(* CODESYS project Flight Simulator.project

Project tree, tasks and I/O mapping:
  PLC : HX-CP1S08, Hitachi Industrial Equipment Systems Co., Ltd., order no. HX-CP1S08, version 3.5.8.24
      settings: IP Address = '192.168.1.1'
    application Application
      libraries: Unit Conversion Interfaces, * (Intern); Standard, * (System); VisuDialogs, * (System); CAA Device Diagnosis, 3.5.4.0 (CAA Technical Workgroup); CAA Net Base Services, 3.5.8.10 (CAA Technical Workgroup); NetVarUdp, 3.5.17.0 (System); PRO JSON, 1.0.0.13 (Pro Electric)
      task Task (cyclic, interval t#20ms, priority 1, watchdog t#100ms x 1) calls MotionTest4_6Servos, TcpClient
      task EtherCAT_Task (cyclic, interval t#8ms, priority 1) calls nothing
      task VISU_TASK (cyclic, interval 100 ms, priority 31) calls VisuElems.Visu_Prg
      Symbols
      program OPC [ST]
      global variables GVL
      program stoplicht [LD]
      program MotionTest1_1Servo [FBD]
      program MotionTest3_1Servo [ST]
      program MotionTest2_1Servo [ST]
      program MotionTest3_2Servos [ST]
      program MotionTest1_2Servos [FBD]
      program MotionTest3_6Servos [ST]
      program MotionTest4_6Servos [ST]
      visualisation Main
      global variables gvlSetting
      data type ServoData
      program TcpClient [ST]
    Basic : Basic, Hitachi-IES, version 3.5.8.20
      _16_Digital_Input : 16 Digital Input, Hitachi-IES, version 3.4.0.0
          unmapped channels: ReserveWord0Type, ReserveWord0Type, ReserveWord0Type
      _16_Digital_Output : 16 Digital Output, Hitachi-IES, version 3.4.0.0
          output Application.GVL.stopLichtGroen : BOOL  // ReserveWord0Type.Bit0
          output Application.GVL.stopLichtGeel : BOOL  // ReserveWord0Type.Bit1
          output Application.GVL.stopLichtRood : BOOL  // ReserveWord0Type.Bit2
          unmapped channels: ReserveWord0Type, ReserveWord0Type, ReserveWord0Type
      _16_Digital_Input_1 : 16 Digital Input, Hitachi-IES, version 3.4.0.0
          unmapped channels: ReserveWord0Type, ReserveWord0Type, ReserveWord0Type
      _16_Digital_Output_1 : 16 Digital Output, Hitachi-IES, version 3.4.0.0
          unmapped channels: ReserveWord0Type, ReserveWord0Type, ReserveWord0Type
      <Empty>
      <Empty>
      <Empty>
      <Empty>
      <Empty>
      <Empty>
      <Empty>
    EtherCAT_Master : EtherCAT Master, Festo, version 3.5.16.43
        settings: MasterUseLRW = False; SlaveAutoRestart = True; NetworkName = 'eth2'; NetworkName = "eth2"; SelectNetworkByName = False; EnableTaskMessage = False; SrcAddress1 = 42135; SrcAddress2 = 3137775364; EnableSecondAdapter = False; SrcAddress = [16#A4,16#97,16#BB,16#06,16#A7,16#04]; NetworkName = 'eth2'; NetworkName = "eth2"; SelectNetworkByName = False
      servo_drive_1 : CMMT-AS (point to point), Festo, order no. 5340819, 534082x, 813335x, version 3.5.16.41
          settings: EnableExpertSettings = True; Watchdog register 0400 = 2498; Watchdog register 0410 = 3000; Watchdog register 0420 = 1000; Physical Address of the Slave = 1001; FMMU.Global Start Address = 16#02000000; FMMU.Physical Start Address = 16#1000; FMMU.Access = 16#02; FMMU.Global Start Address = 16#01000000; FMMU.Physical Start Address = 16#1100; FMMU.Access = 16#01; FMMU.Global Start Address = 16#00080000; FMMU.Physical Start Address = 16#080D; FMMU.Access = 16#01; DC sync0 cycletime = 8000; DC enable = 1; DC sync0 enable = 1; DC sync0 shift time = 0; DC sync1 cycletime = 8000; DC sync1 enable = 0; DC sync1 factor = 'x 1'; DC sync1 shift time = 0
          unmapped channels: Controlword, Modes of operation, Target position, Profile velocity, Target velocity, Target torque, Velocity offset, Torque offset, ---, Statusword, Modes of operation display, Position actual value, Velocity actual value, Torque actual value, Multiturns actual value, ---
      servo_drive_2 : CMMT-AS (point to point), Festo, order no. 5340819, 534082x, 813335x, version 3.5.16.41
          settings: EnableExpertSettings = True; Watchdog register 0400 = 2498; Watchdog register 0410 = 3000; Watchdog register 0420 = 1000; Physical Address of the Slave = 1002; AutoIncr Address of the Slave = 4294967295; FMMU.Global Start Address = 16#02000018; FMMU.Physical Start Address = 16#1000; FMMU.Access = 16#02; FMMU.Global Start Address = 16#01000012; FMMU.Physical Start Address = 16#1100; FMMU.Access = 16#01; FMMU.Global Start Address = 16#00080000; FMMU.StartBit = 1; FMMU.EndBit = 1; FMMU.Physical Start Address = 16#080D; FMMU.Access = 16#01; DC sync0 cycletime = 8000; DC enable = 1; DC sync0 enable = 1; DC sync0 shift time = 0; DC sync1 cycletime = 8000; DC sync1 enable = 0; DC sync1 factor = 'x 1'; DC sync1 shift time = 0
          unmapped channels: Controlword, Modes of operation, Target position, Profile velocity, Target velocity, Target torque, Velocity offset, Torque offset, ---, Statusword, Modes of operation display, Position actual value, Velocity actual value, Torque actual value, Multiturns actual value, ---
      servo_drive_3 : CMMT-AS (point to point), Festo, order no. 5340819, 534082x, 813335x, version 3.5.16.41
          settings: EnableExpertSettings = True; Watchdog register 0400 = 2498; Watchdog register 0410 = 3000; Watchdog register 0420 = 1000; Physical Address of the Slave = 1002; AutoIncr Address of the Slave = 4294967295; FMMU.Global Start Address = 16#02000018; FMMU.Physical Start Address = 16#1000; FMMU.Access = 16#02; FMMU.Global Start Address = 16#01000012; FMMU.Physical Start Address = 16#1100; FMMU.Access = 16#01; FMMU.Global Start Address = 16#00080000; FMMU.StartBit = 1; FMMU.EndBit = 1; FMMU.Physical Start Address = 16#080D; FMMU.Access = 16#01; DC sync0 cycletime = 8000; DC enable = 1; DC sync0 enable = 1; DC sync0 shift time = 0; DC sync1 cycletime = 8000; DC sync1 enable = 0; DC sync1 factor = 'x 1'; DC sync1 shift time = 0
          unmapped channels: Controlword, Modes of operation, Target position, Profile velocity, Target velocity, Target torque, Velocity offset, Torque offset, ---, Statusword, Modes of operation display, Position actual value, Velocity actual value, Torque actual value, Multiturns actual value, ---
      servo_drive_4 : CMMT-AS (point to point), Festo, order no. 5340819, 534082x, 813335x, version 3.5.16.41
          settings: EnableExpertSettings = True; Watchdog register 0400 = 2498; Watchdog register 0410 = 3000; Watchdog register 0420 = 1000; Physical Address of the Slave = 1002; AutoIncr Address of the Slave = 4294967295; FMMU.Global Start Address = 16#02000018; FMMU.Physical Start Address = 16#1000; FMMU.Access = 16#02; FMMU.Global Start Address = 16#01000012; FMMU.Physical Start Address = 16#1100; FMMU.Access = 16#01; FMMU.Global Start Address = 16#00080000; FMMU.StartBit = 1; FMMU.EndBit = 1; FMMU.Physical Start Address = 16#080D; FMMU.Access = 16#01; DC sync0 cycletime = 8000; DC enable = 1; DC sync0 enable = 1; DC sync0 shift time = 0; DC sync1 cycletime = 8000; DC sync1 enable = 0; DC sync1 factor = 'x 1'; DC sync1 shift time = 0
          unmapped channels: Controlword, Modes of operation, Target position, Profile velocity, Target velocity, Target torque, Velocity offset, Torque offset, ---, Statusword, Modes of operation display, Position actual value, Velocity actual value, Torque actual value, Multiturns actual value, ---
      servo_drive_5 : CMMT-AS (point to point), Festo, order no. 5340819, 534082x, 813335x, version 3.5.16.41
          settings: EnableExpertSettings = True; Watchdog register 0400 = 2498; Watchdog register 0410 = 3000; Watchdog register 0420 = 1000; Physical Address of the Slave = 1002; AutoIncr Address of the Slave = 4294967295; FMMU.Global Start Address = 16#02000018; FMMU.Physical Start Address = 16#1000; FMMU.Access = 16#02; FMMU.Global Start Address = 16#01000012; FMMU.Physical Start Address = 16#1100; FMMU.Access = 16#01; FMMU.Global Start Address = 16#00080000; FMMU.StartBit = 1; FMMU.EndBit = 1; FMMU.Physical Start Address = 16#080D; FMMU.Access = 16#01; DC sync0 cycletime = 8000; DC enable = 1; DC sync0 enable = 1; DC sync0 shift time = 0; DC sync1 cycletime = 8000; DC sync1 enable = 0; DC sync1 factor = 'x 1'; DC sync1 shift time = 0
          unmapped channels: Controlword, Modes of operation, Target position, Profile velocity, Target velocity, Target torque, Velocity offset, Torque offset, ---, Statusword, Modes of operation display, Position actual value, Velocity actual value, Torque actual value, Multiturns actual value, ---
      servo_drive_6 : CMMT-AS (point to point), Festo, order no. 5340819, 534082x, 813335x, version 3.5.16.41
          settings: EnableExpertSettings = True; Watchdog register 0400 = 2498; Watchdog register 0410 = 3000; Watchdog register 0420 = 1000; Physical Address of the Slave = 1002; AutoIncr Address of the Slave = 4294967295; FMMU.Global Start Address = 16#02000018; FMMU.Physical Start Address = 16#1000; FMMU.Access = 16#02; FMMU.Global Start Address = 16#01000012; FMMU.Physical Start Address = 16#1100; FMMU.Access = 16#01; FMMU.Global Start Address = 16#00080000; FMMU.StartBit = 1; FMMU.EndBit = 1; FMMU.Physical Start Address = 16#080D; FMMU.Access = 16#01; DC sync0 cycletime = 8000; DC enable = 1; DC sync0 enable = 1; DC sync0 shift time = 0; DC sync1 cycletime = 8000; DC sync1 enable = 0; DC sync1 factor = 'x 1'; DC sync1 shift time = 0
          unmapped channels: Controlword, Modes of operation, Target position, Profile velocity, Target velocity, Target torque, Velocity offset, Torque offset, ---, Statusword, Modes of operation display, Position actual value, Velocity actual value, Torque actual value, Multiturns actual value, ---
  Device : EHV-CPU1025, Hitachi-IES, order no. EHV-CPU1025, version 3.5.4.11
    application Application
      libraries: Standard, * (System); SysTimeRtc, 3.5.17.0 (System); CAA Net Base Services, 3.5.8.10 (CAA Technical Workgroup); PRO JSON, 1.0.0.11 (Pro Electric)
  libraries: VisuSymbols, 4.1.0.0 (System)
  function block Axis [ST]: init, isReady, setPosition, inError, getPosition, cycle, doMovement, doEnable, doReset, doDisable
  function block FlightSimulator [ST]: init, cycle, inError, safetyStop, doReset, doEnable, doDisable, doSyncMovement, doBullshit, setParameters
  text list GlobalTextList
*)

// PLC/Application/ServoData
TYPE ServoData :
STRUCT
	positions: ARRAY[1..6] OF JSONVAR;
	speeds: ARRAY[1..6] OF JSONVAR;
END_STRUCT
END_TYPE

// PLC/Application/GVL
{attribute 'qualified_only'}
VAR_GLOBAL
	stopLichtRood: BOOL;
	stopLichtGeel: BOOL;
	stopLichtGroen: BOOL;
	
	Axis: ARRAY[1..6] OF AXIS_REF_FESTO;
	resetKnop: BOOL := FALSE;
	enableKnop: BOOL := FALSE;
	nextPositionInput: REAL := 0;
	activateKnop: BOOL;
	bullshitKnop: BOOL;
	FlightSimulator: FlightSimulator;
	test: WSTRING := "Je Moeder";
	
END_VAR

// PLC/Application/gvlSetting
{attribute 'qualified_only'}
VAR_GLOBAL CONSTANT
    gc_uiPort        : UINT := 51223;
    gc_stIpAddr      : NBS.IP_ADDR := (sAddr := '145.48.203.188');
     
    gc_wMaxTelegram  : INT := 250; // Length o the telegram
END_VAR

// PLC/Application/MotionTest4_6Servos
PROGRAM MotionTest4_6Servos
VAR
	init: BOOL := TRUE;
	bullshitTimer: TON;
	iCounter : int;
END_VAR

IF init THEN
	GVL.FlightSimulator.init(
		axis1 := servo_drive_1,
		axis2 := servo_drive_2,
		axis3 := servo_drive_3,
		axis4 := servo_drive_4,
		axis5 := servo_drive_5,
		axis6 := servo_drive_6,
		servoData := tcpClient.servoData
	);
	init := FALSE;
END_IF

IF GVL.resetKnop THEN
	GVL.FlightSimulator.doReset();
END_IF

IF GVL.enableKnop THEN
	GVL.FlightSimulator.doEnable();
ELSE
	GVL.FlightSimulator.doDisable();	
END_IF

GVL.FlightSimulator.setParameters(tcpClient.servoData.positions, tcpClient.servoData.speeds);



IF GVL.activateKnop THEN
	//GVL.FlightSimulator.doSyncMovement(position := GVL.nextPositionInput);
	//GVL.FlightSimulator.setParameters(tcpClient.servoData.positions, tcpClient.servoData.speeds);
END_IF

IF GVL.bullshitKnop THEN
	IF bullshitTimer.Q THEN
		GVL.FlightSimulator.doBullshit();
	END_IF
	bullshitTimer(IN:= NOT bullshitTimer.Q, PT := T#0.333S);
END_IF

FOR iCounter := 1 TO 6 BY 1 DO
	GVL.FlightSimulator.currentPositions[iCounter].Number := GVL.FlightSimulator.axis[iCounter].getPosition();
END_FOR



GVL.FlightSimulator.cycle();

END_PROGRAM

// FlightSimulator
FUNCTION_BLOCK FlightSimulator
VAR_OUTPUT
	axis: ARRAY[1..6] OF Axis;
END_VAR
VAR
	sinValue: INT;
	servoData: REFERENCE TO ServoData;
	servoPositions : ARRAY[1..6] OF REAL;
	servoVelocities : ARRAY[1..6] OF REAL;
END_VAR
VAR_INPUT
	currentPositions : ARRAY[1..6] OF JSONVAR;
END_VAR

METHOD init : BOOL
VAR_INPUT
	axis1: REFERENCE TO AXIS_REF_FESTO;
	axis2: REFERENCE TO AXIS_REF_FESTO;
	axis3: REFERENCE TO AXIS_REF_FESTO;
	axis4: REFERENCE TO AXIS_REF_FESTO;
	axis5: REFERENCE TO AXIS_REF_FESTO;
	axis6: REFERENCE TO AXIS_REF_FESTO;
	servoData: REFERENCE TO ServoData;
END_VAR
THIS^.axis[1].init(axis1);
THIS^.axis[2].init(axis2);
THIS^.axis[3].init(axis3);
THIS^.axis[4].init(axis4);
THIS^.axis[5].init(axis5);
THIS^.axis[6].init(axis6);
THIS^.servoData REF= servoData;
END_METHOD

METHOD cycle : BOOL
VAR_INPUT
END_VAR
VAR
	iCounter: UINT;
END_VAR
// If any Axis is in error stop all axis.
IF THIS^.inError() THEN
	THIS^.safetyStop();
END_IF

FOR iCounter := 1 TO 6 BY 1 DO
	IF GVL.activateKnop THEN
		Axis[iCounter].doMovement(position := THIS^.servoPositions[iCounter], velocity := THIS^.servoVelocities[iCounter]);
	END_IF;
END_FOR

// Cycle Axis classes
FOR iCounter := 1 TO 6 BY 1 DO
	THIS^.axis[iCounter].cycle();
END_FOR
END_METHOD

METHOD inError : BOOL
VAR
	iCounter: UINT;
END_VAR
FOR iCounter := 1 TO 6 BY 1 DO
	IF THIS^.axis[iCounter].inError() THEN
		inError := TRUE;
	END_IF
END_FOR
END_METHOD

METHOD safetyStop : BOOL
VAR
	iCounter: UINT;
END_VAR
FOR iCounter := 1 TO 6 BY 1 DO
	Axis[iCounter].doDisable();
END_FOR
END_METHOD

METHOD doReset : BOOL
VAR_INPUT
END_VAR
VAR
	iCounter: UINT;
END_VAR
FOR iCounter := 1 TO 6 BY 1 DO
	Axis[iCounter].doReset();
END_FOR
END_METHOD

METHOD doEnable : BOOL
VAR_INPUT
END_VAR
VAR
	iCounter: INT;
END_VAR
FOR iCounter := 1 TO 6 BY 1 DO
	Axis[iCounter].doEnable();
END_FOR
doEnable := TRUE;
END_METHOD

METHOD doDisable : BOOL
VAR_INPUT
END_VAR
VAR
	iCounter: INT;
END_VAR
FOR iCounter := 1 TO 6 BY 1 DO
	Axis[iCounter].doDisable();
END_FOR
doDisable := TRUE;
END_METHOD

METHOD doSyncMovement : BOOL
VAR_INPUT
	position: REAL;
END_VAR
VAR
	iCounter: INT;
END_VAR
// Only do movements when drive is enabled
FOR iCounter := 1 TO 6 BY 1 DO
	THIS^.axis[iCounter].doMovement(position := position, velocity := 200);
END_FOR
DoSyncMovement := TRUE;	// return
END_METHOD

METHOD doBullshit : BOOL
VAR_INPUT
END_VAR
VAR
	iCounter: INT;
	newPosition: REAL;
END_VAR
FOR iCounter := 1 TO 6 BY 1 DO
	THIS^.sinValue := THIS^.sinValue + 15;
	newPosition := 200.0 + (200.0 * SIN(THIS^.sinValue));
	THIS^.axis[iCounter].doMovement(position := newPosition, velocity := 200);
END_FOR
END_METHOD

METHOD setParameters : BOOL
VAR
	iCounter: INT;
END_VAR
VAR_INPUT
	positions : ARRAY[1..6] OF JSONVAR;
	speeds : ARRAY[1..6] OF JSONVAR;
END_VAR
FOR iCounter := 1 TO 6 BY 1 DO
	THIS^.servoPositions[iCounter] := positions[iCounter].Number;
	THIS^.servoVelocities[iCounter] := speeds[iCounter].Number;
END_FOR
END_METHOD

END_FUNCTION_BLOCK

// Axis
FUNCTION_BLOCK Axis
VAR
	MC_Power: MC_Power_Festo;
	MC_Reset: MC_Reset_Festo;
	MC_MoveAbsolute: MC_MoveAbsolute_Festo;
	MC_ReadActualPosition: MC_ReadActualPosition_Festo;
	MC_ReadStatus: MC_ReadStatus_Festo;
	
	axis: REFERENCE TO AXIS_REF_FESTO;
	done: BOOL := FALSE;
	error: BOOL := FALSE;
	enable: BOOL := FALSE;
	activate: BOOL := FALSE;
	reset: BOOL := FALSE;
	position: REAL := 0;
	velocity: REAL := 200;
	acceleration: REAL := 5000;
	deceleration: REAL := 5000;
	jerk: REAL := 15000;
END_VAR

METHOD init : BOOL
VAR_INPUT
	axis : REFERENCE TO AXIS_REF_FESTO;
END_VAR
// This function references the servo drive to the instance of the function block.
THIS^.axis REF= axis;
END_METHOD

METHOD isReady : BOOL
VAR_INPUT
END_VAR
isReady := THIS^.done;
END_METHOD

METHOD setPosition : BOOL
VAR_INPUT
	position: REAL;
END_VAR
THIS^.position := position;
END_METHOD

METHOD inError : BOOL
VAR_INPUT
END_VAR
inError := THIS^.error;
END_METHOD

METHOD getPosition : REAL
VAR_INPUT
END_VAR
getPosition := THIS^.MC_ReadActualPosition.Position;
END_METHOD

METHOD cycle : BOOL
VAR_INPUT
END_VAR
THIS^.MC_Power(
	axis := THIS^.axis,
	enable := THIS^.enable
);

THIS^.MC_Reset(
	axis := THIS^.axis,
	Execute :=THIS^.reset
);

// Reset the reset variable
IF THIS^.MC_Reset.Done AND THIS^.reset THEN
	THIS^.reset := FALSE;
END_IF

THIS^.MC_MoveAbsolute(
	axis := THIS^.axis,
	Execute := THIS^.activate,
	ContinuousUpdate := FALSE,
	position := THIS^.position,
	velocity := THIS^.velocity,
	acceleration := THIS^.acceleration,
	deceleration := THIS^.deceleration,
	jerk := THIS^.jerk
);

// Reset the activate variable
IF THIS^.MC_MoveAbsolute.Done THEN
	THIS^.activate := FALSE;
	THIS^.done := TRUE;
END_IF

THIS^.MC_ReadActualPosition(
	axis := THIS^.axis,
	Enable := TRUE
);

THIS^.error := THIS^.MC_Power.Error OR THIS^.MC_MoveAbsolute.Error;

//MC_ReadStatus(THIS^.axis);
END_METHOD

METHOD doMovement : BOOL
VAR_INPUT
	velocity: REAL;
	position: REAL;
END_VAR
// Only do movements when drive is enabled
IF THIS^.enable THEN
	THIS^.position := position;
	THIS^.velocity := velocity;
	THIS^.activate := TRUE;
	DoMovement := TRUE;	// return
ELSE
	DoMovement := FALSE;	// return
END_IF;
END_METHOD

METHOD doEnable : BOOL
// Only allow enable when not in error
IF NOT THIS^.inError() THEN
	THIS^.enable := TRUE;
	doEnable := TRUE;
ELSE
	doEnable := FALSE;
END_IF
END_METHOD

METHOD doReset
THIS^.reset := TRUE;
END_METHOD

METHOD doDisable : BOOL
VAR_INPUT
END_VAR
// Allow disable at any time
THIS^.enable := FALSE;
doDisable := TRUE;
END_METHOD

END_FUNCTION_BLOCK

// PLC/Application/TcpClient
PROGRAM TcpClient
VAR
    fbTcpClient   : NBS.TCP_Client;
    fbTcpRead     : NBS.TCP_Read;
    fbTcpWrite    : NBS.TCP_Write;
 
	received      : STRING;
	sent          : STRING;
	parseJSON     : JSON_TO_STRUCT;
	composeJSON   : STRUCT_TO_JSON;
	servoData     : ServoData;
 
    udiVal        : UDINT;
    pudiVal       : POINTER TO BYTE;
    iIndex        : INT;
    xConnect      : BOOL;
 
    xRead         : BOOL := TRUE;
    xMissingAck   : BOOL;
    udiResult     : UDINT;
    udiLastAck    : UDINT;
    udiNow        : UDINT;
    udiRead       : UDINT;
END_VAR

fbTcpClient(xEnable := xConnect, ipAddr := gvlSetting.gc_stIpAddr, uiPort := gvlSetting.gc_uiPort, udiTimeOut := 0);

IF NOT fbTcpWrite.xBusy THEN
	IF NOT composeJSON.Busy THEN
		composeJSON(
		Execute:= TRUE,
		JSONString:= ADR(sent), 
		JSONStringSize:= SIZEOF(sent),
		JSONVars:= ADR(GVL.FlightSimulator.currentPositions),
		NumberOfVars:= SIZEOF(GVL.FlightSimulator.currentPositions) / SIZEOF(JSONVAR)
		);	
	ELSIF composeJSON.Done THEN
		fbTcpWrite(xExecute := xConnect, hConnection := fbTcpClient.hConnection, udiTimeOut := 0, szSize := SIZEOF(sent), pData := ADR(sent));
	END_IF
ELSIF fbTcpWrite.xDone THEN
	fbTcpWrite(xExecute := FALSE);
	composeJSON(Execute := FALSE);	
END_IF

IF NOT fbTcpRead.xBusy THEN
	fbTcpRead(xEnable := xRead AND xConnect, hConnection := fbTcpClient.hConnection, szSize := SIZEOF(received), pData := ADR(received), szCount => udiRead);
	IF fbTcpRead.xReady THEN
		parseJSON(	
		Execute := TRUE,
		JSONString:= ADR(received), 
		JSONStringSize:= SIZEOF(received),
		JSONVars:= ADR(servoData),
		NumberOfVars:= SIZEOF(servoData) / SIZEOF(JSONVAR)
		);
		IF parseJSON.Done THEN
			parseJSON(Execute := FALSE);
		END_IF
	END_IF
END_IF
 
IF NOT fbTcpClient.xActive AND NOT fbTcpClient.xBusy AND NOT fbTcpClient.xDone THEN
    xConnect := TRUE;
ELSIF fbTcpClient.xDone THEN
    xConnect := FALSE;
END_IF

END_PROGRAM

// PLC/Application/OPC
PROGRAM OPC
VAR
	enable : BOOL := FALSE;
	count : INT := 0;
END_VAR

IF enable THEN
	count := count + 1;
END_IF

END_PROGRAM

// PLC/Application/stoplicht
PROGRAM stoplicht
VAR
	timer_1: TON;
	timer_2: TON;
	counter_1: CTU;
END_VAR

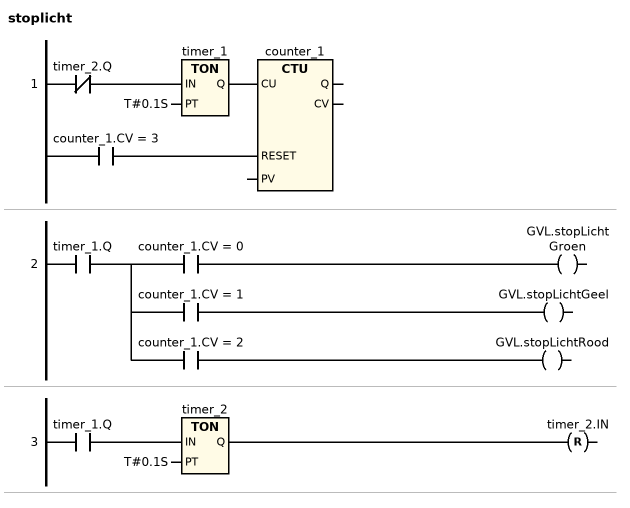
// NETWORK 1
timer_1(IN := NOT timer_2.Q, PT := T#0.1S); // TON
counter_1(CU := timer_1.Q, RESET := counter_1.CV = 3); // CTU

// NETWORK 2
GVL.stopLichtGroen := timer_1.Q AND (counter_1.CV = 0);
GVL.stopLichtGeel := timer_1.Q AND (counter_1.CV = 1);
GVL.stopLichtRood := timer_1.Q AND (counter_1.CV = 2);

// NETWORK 3
timer_2(IN := timer_1.Q, PT := T#0.1S); // TON
timer_2.IN R= timer_2.Q;

END_PROGRAM

// PLC/Application/MotionTest1_1Servo
PROGRAM MotionTest1_1Servo
VAR
	MC_Power: MC_Power_Festo;
	MC_Reset: MC_Reset_Festo;
	MC_MoveAbsolute: MC_MoveAbsolute_Festo;
	Pos: REAL := 0;
	Vel: REAL := 400;
	Acc: REAL := 5000;
	Dec: REAL := 5000;
	Jerk: REAL := 150000;
	Active: BOOL := FALSE;
	Reset: BOOL := FALSE;
	Power: BOOL := FALSE;
	Done: BOOL;
END_VAR
VAR // added by the converter: edge detectors and wires of the graphical bodies
    _w1, _w2 : BOOL;
END_VAR

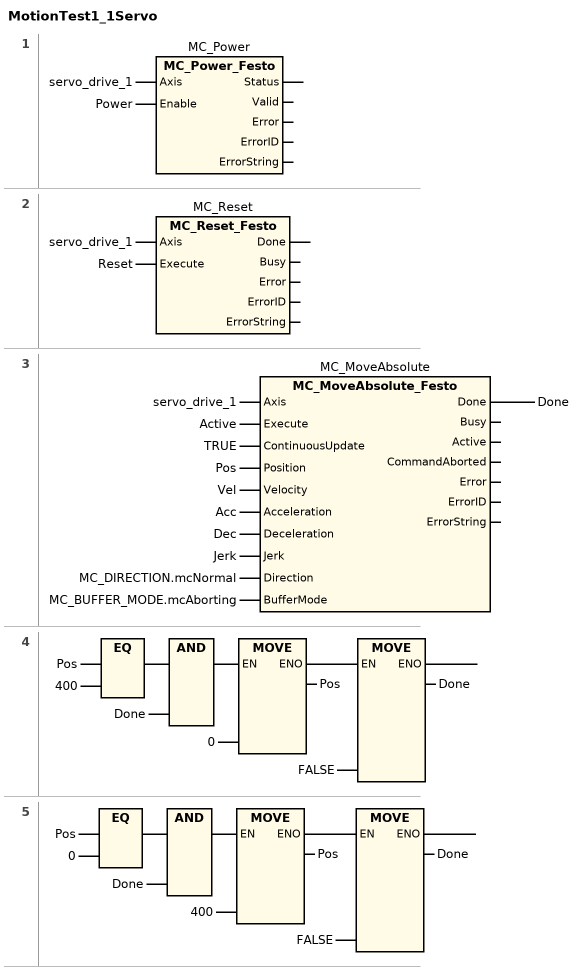
// NETWORK 1
MC_Power(Axis := servo_drive_1, Enable := Power); // MC_Power_Festo

// NETWORK 2
MC_Reset(Axis := servo_drive_1, Execute := Reset); // MC_Reset_Festo

// NETWORK 3
MC_MoveAbsolute(
    Axis := servo_drive_1,
    Execute := Active,
    ContinuousUpdate := TRUE,
    Position := Pos,
    Velocity := Vel,
    Acceleration := Acc,
    Deceleration := Dec,
    Jerk := Jerk,
    Direction := MC_DIRECTION.mcNormal,
    BufferMode := MC_BUFFER_MODE.mcAborting); // MC_MoveAbsolute_Festo
Done := MC_MoveAbsolute.Done;

// NETWORK 4
_w1 := Pos = 400 AND Done;
IF _w1 THEN Pos := 0; END_IF
IF _w1 THEN Done := FALSE; END_IF

// NETWORK 5
_w2 := Pos = 0 AND Done;
IF _w2 THEN Pos := 400; END_IF
IF _w2 THEN Done := FALSE; END_IF

END_PROGRAM

// PLC/Application/MotionTest3_1Servo
PROGRAM MotionTest3_1Servo

VAR
	Pos: REAL := 0;
	Vel: REAL := 400;
	Acc: REAL := 5000;
	Dec: REAL := 5000;
	Jerk: REAL := 150000;
	Active: BOOL := FALSE;
	Power: BOOL := FALSE;
	Done: BOOL;
	init: BOOL := TRUE;
	reset: BOOL := FALSE;
	Axis: Axis;
	inError: BOOL;
END_VAR

//MC_Power(Axis:=servo_drive_1, Enable:=Power, Error => inError);
//MC_Reset(Axis:=servo_drive_1, Execute:=reset, Error => inError);

//MC_MoveAbsolute(Axis:=servo_drive_1, Execute:=Active, ContinuousUpdate:=TRUE, Position:=Pos, Velocity:=Vel, Acceleration:=Acc, Deceleration:=Dec, Jerk:=Jerk);
IF init THEN
	Axis.init(Axis := servo_drive_1);
END_IF

IF Axis.getPosition() >= 399 THEN
	Axis.setPosition(Position := 0);
END_IF

IF Axis.getPosition() <= 1 THEN
	Axis.setPosition(Position := 400);
END_IF

Axis.cycle();

END_PROGRAM

// PLC/Application/MotionTest2_1Servo
PROGRAM MotionTest2_1Servo

VAR
	MC_Power: MC_Power_Festo;
	MC_Reset: MC_Reset_Festo;
	MC_MoveAbsolute: MC_MoveAbsolute_Festo;
	MC_ReadActualPosition: MC_ReadActualPosition_Festo;
	MC_ReadStatus: MC_ReadStatus_Festo;
	Pos: REAL := 0;
	Vel: REAL := 400;
	Acc: REAL := 5000;
	Dec: REAL := 5000;
	Jerk: REAL := 150000;
	Active: BOOL := FALSE;
	Power: BOOL := FALSE;
	Done: BOOL;
	init: BOOL := TRUE;
	reset: BOOL := FALSE;
	Axis: AXIS_REF_FESTO;
	inError: BOOL;
END_VAR

MC_Power(Axis:=servo_drive_1, Enable:=Power, Error => inError);
MC_Reset(Axis:=servo_drive_1, Execute:=reset, Error => inError);

MC_MoveAbsolute(Axis:=servo_drive_1, Execute:=Active, ContinuousUpdate:=TRUE, Position:=Pos, Velocity:=Vel, Acceleration:=Acc, Deceleration:=Dec, Jerk:=Jerk);

END_PROGRAM

// PLC/Application/MotionTest3_2Servos
PROGRAM MotionTest3_2Servos

VAR
	Pos: REAL := 0;
	Vel: REAL := 400;
	Acc: REAL := 5000;
	Dec: REAL := 5000;
	Jerk: REAL := 150000;
	Active: BOOL := FALSE;
	Power: BOOL := FALSE;
	Done: BOOL;
	init: BOOL := TRUE;
	reset: BOOL := FALSE;
	Axis2: Axis;
	Axis1: Axis;
	inError: BOOL;
END_VAR

IF init THEN
	Axis1.init(Axis := servo_drive_1);
	Axis2.init(Axis := servo_drive_2);
END_IF

IF Axis1.getPosition() >= 399 THEN
	Axis1.setPosition(Position := 0);
END_IF

IF Axis1.getPosition() <= 1 THEN
	Axis1.setPosition(Position := 400);
END_IF

IF Axis2.getPosition() >= 399 THEN
	Axis2.setPosition(Position := 0);
END_IF

IF Axis2.getPosition() <= 1 THEN
	Axis2.setPosition(Position := 400);
END_IF

Axis1.cycle();
Axis2.cycle();

END_PROGRAM

// PLC/Application/MotionTest1_2Servos
PROGRAM MotionTest1_2Servos
VAR
	MC_Power_Festo_0: MC_Power_Festo;
	MC_Reset_Festo_0: MC_Reset_Festo;
	MC_MoveAbsolute_Festo_0: MC_MoveAbsolute_Festo;
	Pos: REAL := 0;
	Vel: REAL := 400;
	Acc: REAL := 5000;
	Dec: REAL := 5000;
	Jerk: REAL := 150000;
	Active2: BOOL := FALSE;
	Active: BOOL := FALSE;
	Reset: BOOL := FALSE;
	Power: BOOL := FALSE;
	Power2: BOOL := FALSE;
	Done: BOOL;
	MC_Power_Festo_1: MC_Power_Festo;
	MC_Reset_Festo_1: MC_Reset_Festo;
	MC_MoveAbsolute_Festo_1: MC_MoveAbsolute_Festo;
END_VAR
VAR // added by the converter: edge detectors and wires of the graphical bodies
    _w1, _w2 : BOOL;
END_VAR

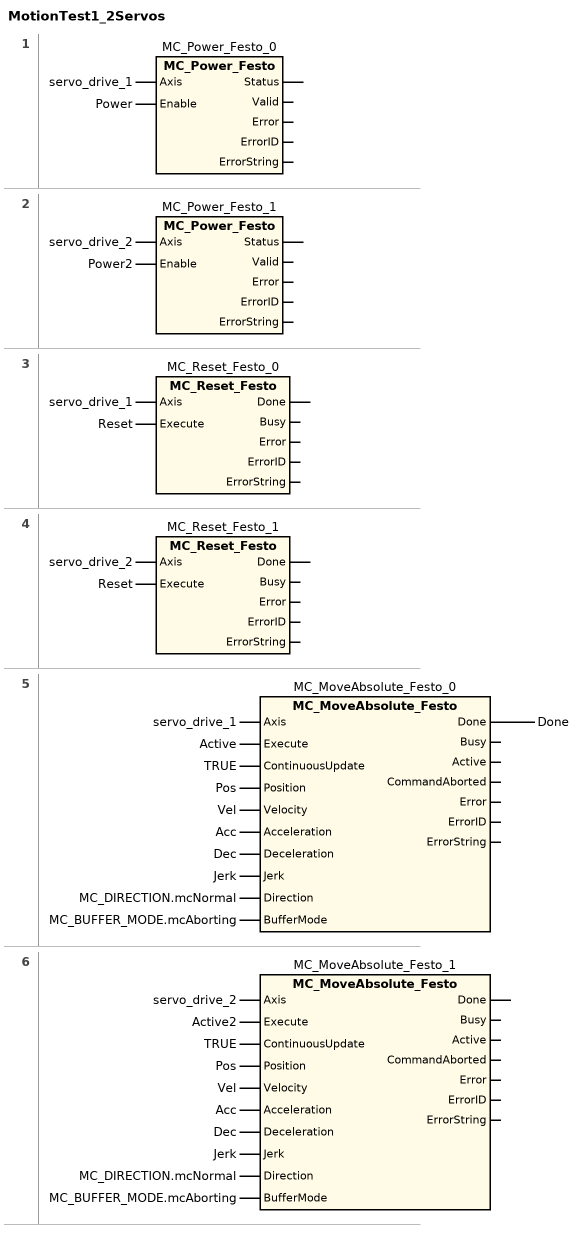
// NETWORK 1
MC_Power_Festo_0(Axis := servo_drive_1, Enable := Power); // MC_Power_Festo

// NETWORK 2
MC_Power_Festo_1(Axis := servo_drive_2, Enable := Power2); // MC_Power_Festo

// NETWORK 3
MC_Reset_Festo_0(Axis := servo_drive_1, Execute := Reset); // MC_Reset_Festo

// NETWORK 4
MC_Reset_Festo_1(Axis := servo_drive_2, Execute := Reset); // MC_Reset_Festo

// NETWORK 5
MC_MoveAbsolute_Festo_0(
    Axis := servo_drive_1,
    Execute := Active,
    ContinuousUpdate := TRUE,
    Position := Pos,
    Velocity := Vel,
    Acceleration := Acc,
    Deceleration := Dec,
    Jerk := Jerk,
    Direction := MC_DIRECTION.mcNormal,
    BufferMode := MC_BUFFER_MODE.mcAborting); // MC_MoveAbsolute_Festo
Done := MC_MoveAbsolute_Festo_0.Done;

// NETWORK 6
MC_MoveAbsolute_Festo_1(
    Axis := servo_drive_2,
    Execute := Active2,
    ContinuousUpdate := TRUE,
    Position := Pos,
    Velocity := Vel,
    Acceleration := Acc,
    Deceleration := Dec,
    Jerk := Jerk,
    Direction := MC_DIRECTION.mcNormal,
    BufferMode := MC_BUFFER_MODE.mcAborting); // MC_MoveAbsolute_Festo

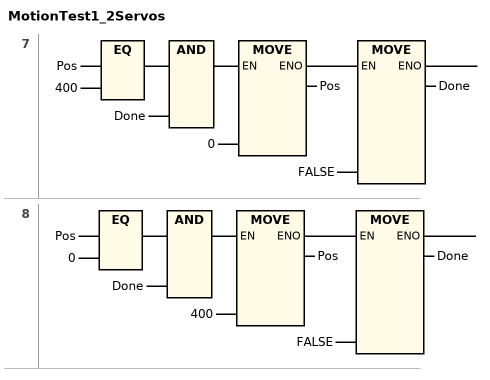
// NETWORK 7
_w1 := Pos = 400 AND Done;
IF _w1 THEN Pos := 0; END_IF
IF _w1 THEN Done := FALSE; END_IF

// NETWORK 8
_w2 := Pos = 0 AND Done;
IF _w2 THEN Pos := 400; END_IF
IF _w2 THEN Done := FALSE; END_IF

END_PROGRAM

// PLC/Application/MotionTest3_6Servos
PROGRAM MotionTest3_6Servos

VAR
	Pos: REAL := 0;
	Vel: REAL := 200;
	Acc: REAL := 5000;
	Dec: REAL := 5000;
	Jerk: REAL := 150000;
	Activate: BOOL := FALSE;
	Enable: BOOL := FALSE;
	Done: BOOL;
	init: BOOL := TRUE;
	reset: BOOL := FALSE;
	inError: BOOL;
	Axis: ARRAY[1..6] OF Axis;
	iCounter: INT;
END_VAR

IF init THEN
	Axis[1].init(servo_drive_1);
	Axis[2].init(servo_drive_2);
	Axis[3].init(servo_drive_3);
	Axis[4].init(servo_drive_4);
	Axis[5].init(servo_drive_5);
	Axis[6].init(servo_drive_6);
	init := FALSE;
END_IF

FOR iCounter := 1 TO 6 BY 1 DO
	Axis[iCounter].doReset();
END_FOR

IF NOT inError THEN
	FOR iCounter := 1 TO 6 BY 1 DO
		Axis[iCounter].doMovement(Pos, Vel);
	END_FOR
	
	IF Enable THEN
		FOR iCounter := 1 TO 6 BY 1 DO
			Axis[iCounter].doEnable();
		END_FOR
	END_IF
END_IF

FOR iCounter := 1 TO 6 BY 1 DO
	IF Axis[iCounter].inError() THEN
		inError := TRUE;
	END_IF
END_FOR

IF inError THEN
	Axis[iCounter].doDisable();
END_IF

FOR iCounter := 1 TO 6 BY 1 DO
	Axis[iCounter].cycle();
END_FOR

END_PROGRAM

// PLC/Application/Main
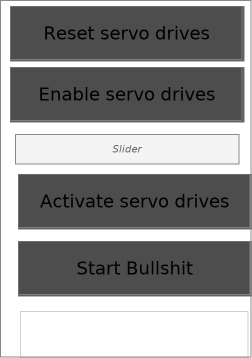
VISUALIZATION Main  // 252x358
    Button (10,6 234x55), "Reset servo drives"
        tap GVL.resetKnop
    Button (10,67 234x55), "Enable servo drives"
        toggle GVL.enableKnop
    Slider (15,134 224x30), variable: GVL.nextPositionInput, scale 0..400
    Button (18,174 234x55), "Activate servo drives"
        toggle GVL.activateKnop
    Button (18,241 234x55), "Start Bullshit"
        toggle GVL.bullshitKnop
    Textfield (20,311 228x47), text variable: GVL.test
END_VISUALIZATION
